PROGRAM P_DelayedLight_Test_ST
VAR
	fbDelayedLight		:	FB_DelayedLight;
	bOn					:	BOOL;
	bOff				:	BOOL;
	bControlLevel		:	BOOL;	
END_VAR

fbDelayedLight();

IF (bOn) THEN
	fbDelayedLight.M_On();
	bOn := FALSE;
END_IF
IF (bOff) THEN
	fbDelayedLight.M_Off();
	bOff := FALSE;
END_IF

bControlLevel := fbDelayedLight.bControlLevel;

END_PROGRAM

(* stored: Version 1.1.0.1, ProductVersion 3.1.0.23
   POU P_DelayedLight_Test_ST: Id {e8ff1aaf-450c-4f38-a1b0-b04587cc28eb} *)
